PROGRAM IO_Map
VAR
	
	
	
	AI3 AT %I*: INT;
END_VAR


//---------------------------------------------	
// EK 1818

	bControlOn				  :=  DI1_1;
	bTopPreserCmdUp           :=  DI1_2;
	bTopPreserCmdDown         :=  DI1_3;
	bCycleStartCmd            :=  DI1_4;
	bCycleStopCmd             :=  DI1_5;
	bCylinderCmdUp            :=  DI1_6;
	bCylinderCmdDown          :=  DI1_7;
	bHydraulicUnitCmdStart    :=  DI1_8;

	
	DO1_1:=bLedHydraulicUnitOn;
	DO1_2;
	DO1_3;
	DO1_4;
//--------------------------------------------	
// EL 4374	
	nHydraulicPressureRaw		:=  AI_1; //{mA]0.004=0bar/0.020=400bar
	nCylinderPositionRaw    	:=  AI_2; //[mA]0.004=0mm/0.020=125mm
	AO_1						:=nHydraulicPressureOut0_10V   	; 
	                          		AO_2;
//--------------------------------------------
	AI3;									
//--------------------------------------------
// EL 1008	
	 bHydraulicUnitRunning		:=  DI2_1;
	 bTopPreserClosed           :=  DI2_2;
	 bTopPreserMotorOk          :=  DI2_3;
	 bHydraulicUnitMotorOk      :=  DI2_4;
	 bHydraulicUnitCmdStop      :=  DI2_5;
	 bOilLevelOk                :=  DI2_6;
	 bEstopOk                   :=  DI2_7;
	                                DI2_8;
	
//--------------------------------------------
//EL 2008
	DO2_1:=bTopPreserUp ;
	DO2_2:=bTopPreserDown ;
	DO2_3:=bHydraulicUintOn ;
	DO2_4:=bLedCycleOn ;
	DO2_5:=bReliefValveOn ;
	DO2_6:=bCylinderValveUp ;
	DO2_7:=bCylinderValveDown ;
	DO2_8:=bProportionalValveEnable AND  .bCylinderValveUp ;

END_PROGRAM

(* stored: Version 1.1.0.1, ProductVersion 3.1.4024.16
   POU IO_Map: Id {d5cb3b4f-f901-4858-a3fa-b8e4dc11805b}, SpecialFunc None *)
